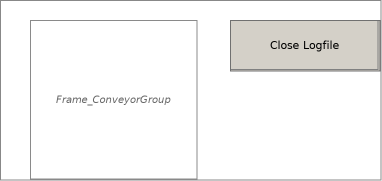
VISUALIZATION VISU_CONVEYOR_TEST  // 382x181
    Frame (30,20 167x159)
        shows Frame_ConveyorGroup(vio_fbConveyor1 := CONVEYOR_TEST.aConveyors[1], vio_fbConveyor2 := CONVEYOR_TEST.aConveyors[2], vio_fbConveyor3 := CONVEYOR_TEST.aConveyors[3], vio_fbConveyor4 := CONVEYOR_TEST.aConveyors[4], vio_fbConveyor5 := CONVEYOR_TEST.aConveyors[5], vio_fbConveyor6 := CONVEYOR_TEST.aConveyors[6], vio_fbConveyor7 := CONVEYOR_TEST.aConveyors[7], vio_fbConveyor8 := CONVEYOR_TEST.aConveyors[8])
    Button (230,20 150x51), "Close Logfile"
        tap CONVEYOR_TEST.bCloseFile
END_VISUALIZATION

(* stored: Version 1.1.0.1, ProductVersion 3.1.4022.16
   Visu VISU_CONVEYOR_TEST: Id {51cad7f7-0fd7-436b-bfaa-c9fd16659817} *)
